PROGRAM PRG_TerminalMapping
VAR
    uiIndexPositionCode : UINT;
END_VAR

// ============================================================================
// TE1108 Silicone Station - EPLAN Rev 1.0 terminal mapping
//
// ReadInputs:
//   EtherCAT inputs and TwinSAFE aliases -> GVL_IO.stInputs
//
// WriteOutputs:
//   GVL_IO.stOutputs -> EtherCAT outputs and TwinSAFE request aliases
//
// Execution order:
//   PRG_TerminalMapping.ReadInputs();
//   application logic;
//   PRG_TerminalMapping.WriteOutputs();
// ============================================================================

METHOD PUBLIC ReadInputs
VAR_INPUT
END_VAR
// ---------------------------------------------------------------------------
// Term 4 - EL1918(EPLAN page 11)
// ---------------------------------------------------------------------------
GVL_IO.stInputs.bEmergencyStopChannel1 			:= GVL_EtherCAT.stTerm4_EL1918.iEL1918_Ch1;
GVL_IO.stInputs.bEmergencyStopChannel2 			:= GVL_EtherCAT.stTerm4_EL1918.iEL1918_Ch2;
GVL_IO.stInputs.bMainDoorChannel1 				:= GVL_EtherCAT.stTerm4_EL1918.iEL1918_Ch4;
GVL_IO.stInputs.bMainDoorChannel2 				:= GVL_EtherCAT.stTerm4_EL1918.iEL1918_Ch5;
GVL_IO.stInputs.bMainDoorFeedback 				:= GVL_EtherCAT.stTerm4_EL1918.iEL1918_Ch6;
GVL_IO.stInputs.bMs6FeedbackOk 					:= GVL_EtherCAT.stTerm4_EL1918.iEL1918_Ch7;
GVL_IO.stInputs.bAirExhausted 					:= GVL_EtherCAT.stTerm4_EL1918.iEL1918_Ch8;

// ---------------------------------------------------------------------------
// Term 5 - EL1918(EPLAN page 12)
// ---------------------------------------------------------------------------
GVL_IO.stInputs.bTouchButtonleft 				:= GVL_EtherCAT.stTerm5_EL1918.iEL1918_Ch3;
GVL_IO.stInputs.bTouchButtonRight 				:= GVL_EtherCAT.stTerm5_EL1918.iEL1918_Ch4;

GVL_IO.stInputs.bRightFlapChannel1   			:= GVL_EtherCAT.stTerm5_EL1918.iEL1918_Ch5;
GVL_IO.stInputs.bRightFlapChannel2     			:= GVL_EtherCAT.stTerm5_EL1918.iEL1918_Ch6;
GVL_IO.stInputs.bLeftFlapChannel1  				:= GVL_EtherCAT.stTerm5_EL1918.iEL1918_Ch7;
GVL_IO.stInputs.bLeftFlapChannel2  				:= GVL_EtherCAT.stTerm5_EL1918.iEL1918_Ch8;



// ---------------------------------------------------------------------------
// Term 7 - EL1809 (EPLAN page 14)
// ---------------------------------------------------------------------------
GVL_IO.stInputs.bStartButton 					:= GVL_EtherCAT.stTerm7_EL1809.iEL1809_Ch1;
GVL_IO.stInputs.bStopButton 					:= NOT GVL_EtherCAT.stTerm7_EL1809.iEL1809_Ch2;
GVL_IO.stInputs.bUp24VPowerSupplyOk 			:= GVL_EtherCAT.stTerm7_EL1809.iEL1809_Ch3;
GVL_IO.stInputs.bUs24VPowerSupplyOk 			:= GVL_EtherCAT.stTerm7_EL1809.iEL1809_Ch4;
GVL_IO.stInputs.bIvekHeaterControllerAlarm 		:= GVL_EtherCAT.stTerm7_EL1809.iEL1809_Ch5;

GVL_IO.stInputs.bIndexPositionSensor1 			:= GVL_EtherCAT.stTerm7_EL1809.iEL1809_Ch6;
GVL_IO.stInputs.bIndexPositionSensor2 			:= GVL_EtherCAT.stTerm7_EL1809.iEL1809_Ch7;
GVL_IO.stInputs.bIndexPositionSensor3 			:= GVL_EtherCAT.stTerm7_EL1809.iEL1809_Ch8;
GVL_IO.stInputs.bIndexCompletedSensor 			:= GVL_EtherCAT.stTerm7_EL1809.iEL1809_Ch9;
GVL_IO.stInputs.bIndexLocked 					:= GVL_EtherCAT.stTerm7_EL1809.iEL1809_Ch10;
GVL_IO.stInputs.bIndexReady 					:= GVL_EtherCAT.stTerm7_EL1809.iEL1809_Ch11;

GVL_IO.stInputs.bGearboxAssemblyPartPresent 	:= GVL_EtherCAT.stTerm7_EL1809.iEL1809_Ch12;
GVL_IO.stInputs.bReservoirPartPresent 			:= GVL_EtherCAT.stTerm7_EL1809.iEL1809_Ch13;
GVL_IO.stInputs.bRejectChutePartPresent 		:= GVL_EtherCAT.stTerm7_EL1809.iEL1809_Ch14;
GVL_IO.stInputs.bSiliconeMinimumLevelSensor1 	:= GVL_EtherCAT.stTerm7_EL1809.iEL1809_Ch15;
GVL_IO.stInputs.bSiliconeMinimumLevelSensor2 	:= GVL_EtherCAT.stTerm7_EL1809.iEL1809_Ch16;

GVL_IO.stInputs.bBothPartPresent				:= GVL_EtherCAT.stTerm7_EL1809.iEL1809_Ch12 AND GVL_EtherCAT.stTerm7_EL1809.iEL1809_Ch13;

// Position inputs are documented as binary weights 1, 2 and 4.
uiIndexPositionCode := UINT#0;
IF GVL_IO.stInputs.bIndexPositionSensor1 THEN
    uiIndexPositionCode := uiIndexPositionCode + UINT#1;
END_IF
IF GVL_IO.stInputs.bIndexPositionSensor2 THEN
    uiIndexPositionCode := uiIndexPositionCode + UINT#2;
END_IF
IF GVL_IO.stInputs.bIndexPositionSensor3 THEN
    uiIndexPositionCode := uiIndexPositionCode + UINT#4;
END_IF


IF GVL_IO.stInputs.bIndexLocked THEN
    GVL_IO.stInputs.eIndexPosition := UINT_TO_E_TablePosition(uiIndexPositionCode);
ELSE
    GVL_IO.stInputs.eIndexPosition := E_TablePosition.Unknown;
END_IF

// ---------------------------------------------------------------------------
// Term 8 - EL1809 (EPLAN page 15)
// ---------------------------------------------------------------------------

GVL_IO.stInputs.bSiliconeSupportRetracted 					:= 	GVL_EtherCAT.stTerm8_EL1809.iEL1809_Ch1;
GVL_IO.stInputs.bSiliconeSupportExtended 					:= 	GVL_EtherCAT.stTerm8_EL1809.iEL1809_Ch2;
GVL_IO.stInputs.bAssemblySupportRetracted 					:=	GVL_EtherCAT.stTerm8_EL1809.iEL1809_Ch3;
GVL_IO.stInputs.bAssemblySupportExtended 					:=	GVL_EtherCAT.stTerm8_EL1809.iEL1809_Ch4;

// Flipping station feedback - EPLAN page 15
GVL_IO.stInputs.bTransferVerticalMiniSlideRetracted     := GVL_EtherCAT.stTerm8_EL1809.iEL1809_Ch5;
GVL_IO.stInputs.bTransferVerticalMiniSlideExtended      := GVL_EtherCAT.stTerm8_EL1809.iEL1809_Ch6;
GVL_IO.stInputs.bRotaryGripperOpened                    := GVL_EtherCAT.stTerm8_EL1809.iEL1809_Ch7;
GVL_IO.stInputs.bRotaryGripperClosed                    := GVL_EtherCAT.stTerm8_EL1809.iEL1809_Ch8;
GVL_IO.stInputs.bRotaryGripperRotationPick0             := GVL_EtherCAT.stTerm8_EL1809.iEL1809_Ch9;
GVL_IO.stInputs.bRotaryGripperRotationPlace180          := GVL_EtherCAT.stTerm8_EL1809.iEL1809_Ch10;
GVL_IO.stInputs.bSiliconeStationPartPresent 			:=GVL_EtherCAT.stTerm8_EL1809.iEL1809_Ch11;

// ---------------------------------------------------------------------------
// / Term 11 -Analog inputs - raw process values (EPLAN pages 21 and 22)
// ---------------------------------------------------------------------------
GVL_IO.stInputs.uiMainAirPressureRaw 						:= GVL_EtherCAT.stTerm11_EL3058.iEL3058_Ch1;

// ---------------------------------------------------------------------------
// / Term 12 -Analog inputs Voltage
// ---------------------------------------------------------------------------
GVL_IO.stInputs.uiVacuumPressureRaw 						:= GVL_EtherCAT.stTerm12_EL3064.iEL3064_Ch1;
GVL_IO.stInputs.uiExtractionAVacuumPressureRaw				:= GVL_EtherCAT.stTerm12_EL3064.iEL3064_Ch2;
GVL_IO.stInputs.iPartVacuumPressureRaw 						:= GVL_EtherCAT.stTerm12_EL3064.iEL3064_Ch3;

// ---------------------------------------------------------------------------
// / Term 14 -Analog inputs Voltage
// ---------------------------------------------------------------------------
GVL_IO.stInputs.uiSiliconePressureRaw 						:= GVL_EtherCAT.stTerm14_EL3064.iEL3064_Ch2;
GVL_IO.stInputs.uiNozzlePressureRaw 						:= GVL_EtherCAT.stTerm14_EL3064.iEL3064_Ch1;

// ---------------------------------------------------------------------------
// / Term 33 -Analog inputs Voltage
// ---------------------------------------------------------------------------
GVL_IO.stInputs.iIvekHeaterTemperature						:= GVL_EtherCAT.stTerm33_EL3314.iEL3314_Ch1;

// ---------------------------------------------------------------------------
// TwinSAFE -> PLC validated aliases
// ---------------------------------------------------------------------------
GVL_IO.stInputs.bResetButton 								:= GVL_Safety.bResetButtonPressed;
GVL_IO.stInputs.bTwoHandsSafe 								:= GVL_Safety.bTwoHandSafe;
GVL_IO.stInputs.bSafetyOk 									:= GVL_Safety.bSafetyOk;
//GVL_IO.stInputs.bEmergencyStopOk 							:= GVL_Safety.bEmergencyStopOk;
//GVL_IO.stInputs.bMainDoorSafe 								:= GVL_Safety.bMainDoorSafe;
//GVL_IO.stInputs.bLeftFlapSafe 								:= GVL_Safety.bLeftFlapSafe;
//GVL_IO.stInputs.bRightFlapSafe 								:= GVL_Safety.bRightFlapSafe;
//GVL_IO.stInputs.bFlapsSafe 									:= GVL_Safety.bFlapsSafe;
//GVL_IO.stInputs.bFsoeOk 									:= GVL_Safety.bFsoeOk;
//GVL_IO.stInputs.bSafetyLogicOk 								:= GVL_Safety.bSafetyLogicOk;
GVL_IO.stInputs.bAirSupplyOk 								:= GVL_Safety.bAirSupplySafe;
GVL_IO.stInputs.bMainDoorClosed 							:= GVL_Safety.bMainDoorClosed;
GVL_IO.stInputs.bMainDoorLocked 							:= GVL_Safety.bMainDoorLocked;
GVL_IO.stInputs.bMainDoorUnsafe 							:= GVL_Safety.bMainDoorUnsafe;
GVL_IO.stInputs.bMainDoorDiagnosticOk 						:= GVL_Safety.bMainDoorDiagnosticOk;
// GVL_IO.stInputs.bMs6FeedbackOk 								:= GVL_Safety.bMs6FeedbackOk;
// GVL_IO.stInputs.bAirExhausted 								:= GVL_Safety.bAirExhausted;



// =========================================================
// ETHERCAT TERMINAL OPERATIONAL STATUS
// State 8 = EtherCAT OP
// =========================================================

GVL_EtherCAT.stTerm1_EK1100.stTerminalInfo.bTerminalOperational :=
    GVL_EtherCAT.stTerm1_EK1100.stTerminalInfo.nTerminal_State = UINT#8;

GVL_EtherCAT.stTerm2_EL6070.stTerminalInfo.bTerminalOperational :=
    GVL_EtherCAT.stTerm2_EL6070.stTerminalInfo.nTerminal_State = UINT#8;

GVL_EtherCAT.stTerm3_EL6910.stTerminalInfo.bTerminalOperational :=
    GVL_EtherCAT.stTerm3_EL6910.stTerminalInfo.nTerminal_State = UINT#8;

GVL_EtherCAT.stTerm4_EL1918.stTerminalInfo.bTerminalOperational :=
    GVL_EtherCAT.stTerm4_EL1918.stTerminalInfo.nTerminal_State = UINT#8;

GVL_EtherCAT.stTerm5_EL1918.stTerminalInfo.bTerminalOperational :=
    GVL_EtherCAT.stTerm5_EL1918.stTerminalInfo.nTerminal_State = UINT#8;

GVL_EtherCAT.stTerm6_EL2904.stTerminalInfo.bTerminalOperational :=
    GVL_EtherCAT.stTerm6_EL2904.stTerminalInfo.nTerminal_State = UINT#8;

GVL_EtherCAT.stTerm7_EL1809.stTerminalInfo.bTerminalOperational :=
    GVL_EtherCAT.stTerm7_EL1809.stTerminalInfo.nTerminal_State = UINT#8;

GVL_EtherCAT.stTerm8_EL1809.stTerminalInfo.bTerminalOperational :=
    GVL_EtherCAT.stTerm8_EL1809.stTerminalInfo.nTerminal_State = UINT#8;

GVL_EtherCAT.stTerm9_EL2809.stTerminalInfo.bTerminalOperational :=
    GVL_EtherCAT.stTerm9_EL2809.stTerminalInfo.nTerminal_State = UINT#8;

GVL_EtherCAT.stTerm10_EL2809.stTerminalInfo.bTerminalOperational :=
    GVL_EtherCAT.stTerm10_EL2809.stTerminalInfo.nTerminal_State = UINT#8;

GVL_EtherCAT.stTerm11_EL3058.stTerminalInfo.bTerminalOperational :=
    GVL_EtherCAT.stTerm11_EL3058.stTerminalInfo.nTerminal_State = UINT#8;

GVL_EtherCAT.stTerm12_EL3064.stTerminalInfo.bTerminalOperational :=
    GVL_EtherCAT.stTerm12_EL3064.stTerminalInfo.nTerminal_State = UINT#8;

GVL_EtherCAT.stTerm13_EL9410.stTerminalInfo.bTerminalOperational :=
    GVL_EtherCAT.stTerm13_EL9410.stTerminalInfo.nTerminal_State = UINT#8;

GVL_EtherCAT.stTerm14_EL3064.stTerminalInfo.bTerminalOperational :=
    GVL_EtherCAT.stTerm14_EL3064.stTerminalInfo.nTerminal_State = UINT#8;

GVL_EtherCAT.stTerm15_EL6652.stTerminalInfo.bTerminalOperational :=
    GVL_EtherCAT.stTerm15_EL6652.stTerminalInfo.nTerminal_State = UINT#8;

GVL_EtherCAT.stTerm33_EL3314.stTerminalInfo.bTerminalOperational :=
    GVL_EtherCAT.stTerm33_EL3314.stTerminalInfo.nTerminal_State = UINT#8;
END_METHOD

METHOD PUBLIC WriteOutputs
VAR_INPUT
END_VAR
// ---------------------------------------------------------------------------
// Standard PLC -> TwinSAFE request aliases
// TwinSAFE owns Term 6 EL2904 outputs (air supply and front-door control).
// ---------------------------------------------------------------------------
GVL_Safety.bSafetyRunRequest 					:= GVL_IO.stOutputs.bSafetyRunRequest;
GVL_Safety.bSafetyResetRequest 					:= GVL_IO.stOutputs.bSafetyResetRequest;
GVL_Safety.bAirSupplyEnableRequest 				:= GVL_IO.stOutputs.bAirSupplyEnable;
GVL_Safety.bMainDoorLockRequest 				:= GVL_IO.stOutputs.bMainDoorLockRequest;

// ---------------------------------------------------------------------------
// Safety 
// ---------------------------------------------------------------------------
GVL_Safety.bSafetyErrorAcknowledgementRequest 	:= GVL_IO.stOutputs.bSafetyErrorAcknowledgementRequest;
// ---------------------------------------------------------------------------
// Term 9 - EL2809-0015 (EPLAN page 17)
// ---------------------------------------------------------------------------
GVL_EtherCAT.stTerm9_EL2809.iEL2809_Ch1 		:= GVL_IO.stOutputs.bLedStart;
GVL_EtherCAT.stTerm9_EL2809.iEL2809_Ch2 		:= GVL_IO.stOutputs.bLedReset;
GVL_EtherCAT.stTerm9_EL2809.iEL2809_Ch3 		:= GVL_IO.stOutputs.bLedFail;
GVL_EtherCAT.stTerm9_EL2809.iEL2809_Ch4 		:= GVL_IO.stOutputs.bLedPass;
GVL_EtherCAT.stTerm9_EL2809.iEL2809_Ch5 		:= GVL_IO.stOutputs.bInternalLight;
GVL_EtherCAT.stTerm9_EL2809.iEL2809_Ch6 		:= GVL_IO.stOutputs.bNestLight OR GVL_IO.stOutputs.bExternalLight;
GVL_EtherCAT.stTerm9_EL2809.iEL2809_Ch7 		:= GVL_IO.stOutputs.bVacuumPumpEnable;
GVL_EtherCAT.stTerm9_EL2809.iEL2809_Ch8 		:= GVL_IO.stOutputs.bVacuumAirSolenoid1;
GVL_EtherCAT.stTerm9_EL2809.iEL2809_Ch9 		:= GVL_IO.stOutputs.bVacuumAirSolenoid2;
GVL_EtherCAT.stTerm9_EL2809.iEL2809_Ch10 		:= GVL_IO.stOutputs.bExtractorEnable;
GVL_EtherCAT.stTerm9_EL2809.iEL2809_Ch11 		:= GVL_IO.stOutputs.bSiliconeAirEnable;
GVL_EtherCAT.stTerm9_EL2809.iEL2809_Ch12 		:= FALSE;
GVL_EtherCAT.stTerm9_EL2809.iEL2809_Ch13 		:= FALSE;
GVL_EtherCAT.stTerm9_EL2809.iEL2809_Ch14 		:= FALSE;
GVL_EtherCAT.stTerm9_EL2809.iEL2809_Ch15 		:= FALSE;
GVL_EtherCAT.stTerm9_EL2809.iEL2809_Ch16 		:= FALSE;

// ---------------------------------------------------------------------------
// Term 10 - EL2809-0015 (EPLAN page 19)
// Note the EPLAN order: Ch1 = Port B, Ch2 = Port A.
// ---------------------------------------------------------------------------
GVL_EtherCAT.stTerm10_EL2809.iEL2809_Ch1 		:= GVL_IO.stOutputs.bIndexStopPortB;
GVL_EtherCAT.stTerm10_EL2809.iEL2809_Ch2 		:= GVL_IO.stOutputs.bIndexRotatePortA;
GVL_EtherCAT.stTerm10_EL2809.iEL2809_Ch3 		:= GVL_IO.stOutputs.bSiliconeSupportExtend;
GVL_EtherCAT.stTerm10_EL2809.iEL2809_Ch4 		:= GVL_IO.stOutputs.bSiliconeSupportRetract;
GVL_EtherCAT.stTerm10_EL2809.iEL2809_Ch5 		:= GVL_IO.stOutputs.bAssemblySupportExtend;
GVL_EtherCAT.stTerm10_EL2809.iEL2809_Ch6 		:= GVL_IO.stOutputs.bAssemblySupportRetract;
GVL_EtherCAT.stTerm10_EL2809.iEL2809_Ch7 		:= GVL_IO.stOutputs.bSiliconePinchValve1;
GVL_EtherCAT.stTerm10_EL2809.iEL2809_Ch8 		:= GVL_IO.stOutputs.bSiliconePinchValve2;
GVL_EtherCAT.stTerm10_EL2809.iEL2809_Ch9        := GVL_IO.stOutputs.bTransferVerticalMiniSlideRetract; //GVL_IO.stOutputs.bTransferVerticalMiniSlideExtend;
GVL_EtherCAT.stTerm10_EL2809.iEL2809_Ch10       := GVL_IO.stOutputs.bTransferVerticalMiniSlideExtend; //GVL_IO.stOutputs.bTransferVerticalMiniSlideRetract;
GVL_EtherCAT.stTerm10_EL2809.iEL2809_Ch11       := GVL_IO.stOutputs.bRotaryGripperRotationPlace180; //GVL_IO.stOutputs.bRotaryGripperRotationPick0; //GVL_IO.stOutputs.bRotaryGripperOpen;
GVL_EtherCAT.stTerm10_EL2809.iEL2809_Ch12       := GVL_IO.stOutputs.bRotaryGripperRotationPick0; //GVL_IO.stOutputs.bRotaryGripperRotationPlace180; //GVL_IO.stOutputs.bRotaryGripperClose;
GVL_EtherCAT.stTerm10_EL2809.iEL2809_Ch13       := GVL_IO.stOutputs.bRotaryGripperClose; //GVL_IO.stOutputs.bRotaryGripperOpen; //GVL_IO.stOutputs.bRotaryGripperRotationPick0;
GVL_EtherCAT.stTerm10_EL2809.iEL2809_Ch14       := GVL_IO.stOutputs.bRotaryGripperOpen; //GVL_IO.stOutputs.bRotaryGripperClose; //GVL_IO.stOutputs.bRotaryGripperRotationPlace180;
GVL_EtherCAT.stTerm10_EL2809.iEL2809_Ch15 		:= GVL_IO.stOutputs.bPartVacuumEnable;
GVL_EtherCAT.stTerm10_EL2809.iEL2809_Ch16 		:= FALSE;
END_METHOD

END_PROGRAM

(* stored: Version 1.1.0.1, ProductVersion 3.1.4026.18
   POU PRG_TerminalMapping: Id {7aa70a09-865b-4c80-8264-2867e47e0f23}, SpecialFunc None
   Method ReadInputs: Id {f0a59f2b-b078-4cda-8914-06278c9b0ffc}
   Method WriteOutputs: Id {4e3bd4ad-ac4e-448e-a2a8-70de4747ca16} *)
